% RSLogix 500 project Digital-Rotameter.RSS, saved by version 8.30.00.16 %
PROJECT "UNTITLED"    % processor: Bul.1763 MicroLogix 1100 Series B %

PROGRAM FILES
  LAD 2 "MAIN"  5 rungs

DATA FILES
  O0 OUTPUT  4 elements
  I1 INPUT  6 elements
  S2 STATUS  66 elements
  B3 BINARY  1 elements
  T4 TIMER  2 elements
  C5 COUNTER  1 elements
  R6 CONTROL  1 elements
  N7 INTEGER  1 elements
  F8 FLOAT  3 elements

LADDER 2 "MAIN"
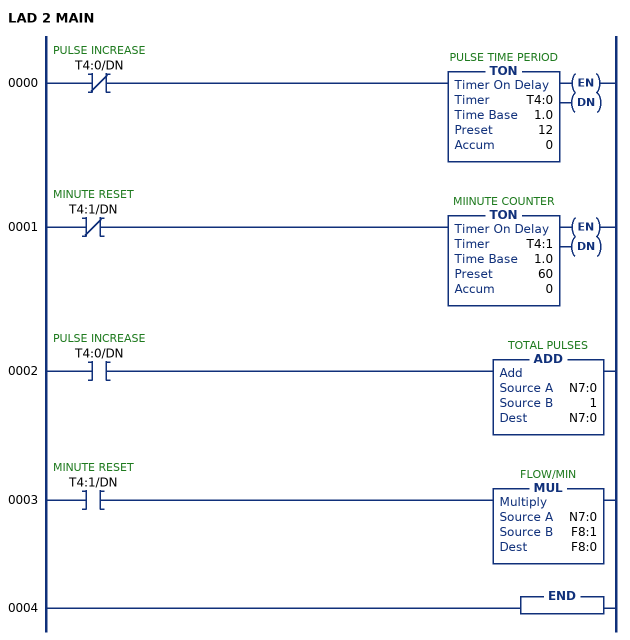
% Rung: 0 %
SOR XIO T4:0/DN TON T4:0 1.0 12 0 EOR
%   T4:0/DN  "PULSE INCREASE" %
%   T4:0  "PULSE TIME PERIOD" %
% Rung: 1 %
SOR XIO T4:1/DN TON T4:1 1.0 60 0 EOR
%   T4:1/DN  "MINUTE RESET" %
%   T4:1  "MIINUTE COUNTER" %
% Rung: 2 %
SOR XIC T4:0/DN ADD N7:0 1 N7:0 EOR
%   T4:0/DN  "PULSE INCREASE" %
%   N7:0  "TOTAL PULSES" %
% Rung: 3 %
SOR XIC T4:1/DN MUL N7:0 F8:1 F8:0 EOR
%   T4:1/DN  "MINUTE RESET" %
%   N7:0  "TOTAL PULSES" %
%   F8:1  "FLOW PER PULSE" %
%   F8:0  "FLOW/MIN" %
% Rung: 4 %
SOR END EOR

DATA TABLE (non-zero values as saved)
DATA T4
% .PRE .ACC %
% T4:0 % 12 0
% T4:1 % 60 0
DATA F8
% F8:0 % 0 6.3 0
